// Mitsubishi GX Works2 project: 시퀀스 부분 반복 회로 예제   PLC: Q03UDV

PROGRAM MAIN
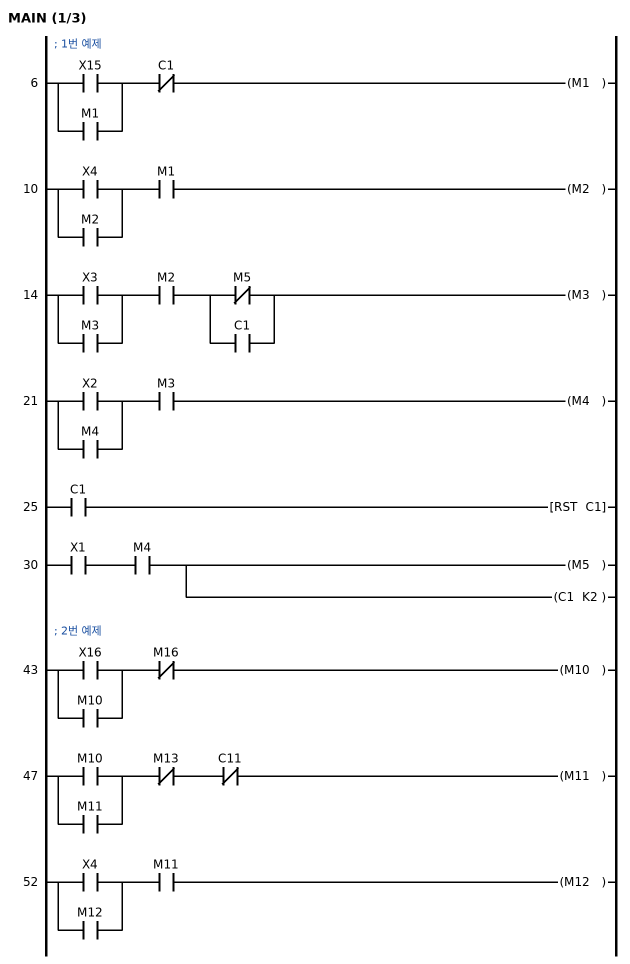
; 1번 예제
6     LD      X15
      OR      M1
      ANI     C1
      OUT     M1
10    LD      X4
      OR      M2
      AND     M1
      OUT     M2
14    LD      X3
      OR      M3
      AND     M2
      LDI     M5
      OR      C1
      ANB
      OUT     M3
21    LD      X2
      OR      M4
      AND     M3
      OUT     M4
25    LD      C1
      RST     C1
30    LD      X1
      AND     M4
      OUT     M5
      OUT     C1 K2
; 2번 예제
43    LD      X16
      OR      M10
      ANI     M16
      OUT     M10
47    LD      M10
      OR      M11
      ANI     M13
      ANI     C11
      OUT     M11
52    LD      X4
      OR      M12
      AND     M11
      OUT     M12
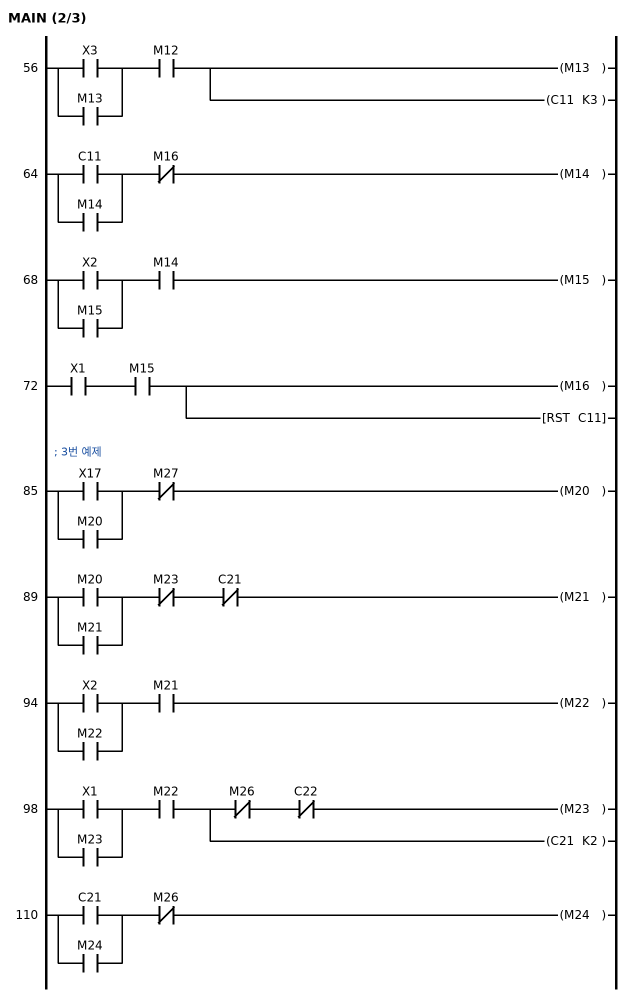
56    LD      X3
      OR      M13
      AND     M12
      OUT     M13
      OUT     C11 K3
64    LD      C11
      OR      M14
      ANI     M16
      OUT     M14
68    LD      X2
      OR      M15
      AND     M14
      OUT     M15
72    LD      X1
      AND     M15
      OUT     M16
      RST     C11
; 3번 예제
85    LD      X17
      OR      M20
      ANI     M27
      OUT     M20
89    LD      M20
      OR      M21
      ANI     M23
      ANI     C21
      OUT     M21
94    LD      X2
      OR      M22
      AND     M21
      OUT     M22
98    LD      X1
      OR      M23
      AND     M22
      MPS
      ANI     M26
      ANI     C22
      OUT     M23
      MPP
      OUT     C21 K2
110   LD      C21
      OR      M24
      ANI     M26
      OUT     M24
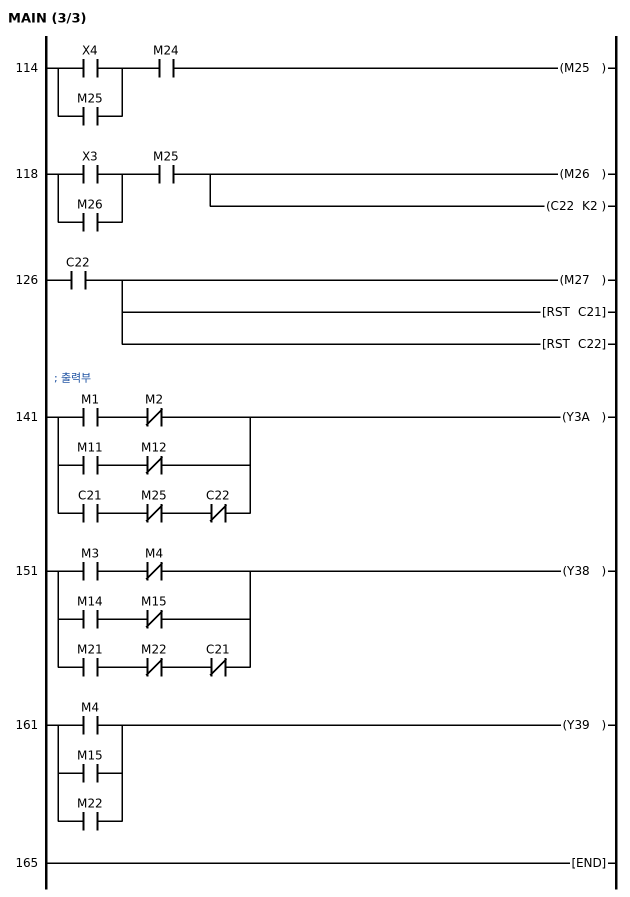
114   LD      X4
      OR      M25
      AND     M24
      OUT     M25
118   LD      X3
      OR      M26
      AND     M25
      OUT     M26
      OUT     C22 K2
126   LD      C22
      OUT     M27
      RST     C21
      RST     C22
; 출력부
141   LD      M1
      ANI     M2
      LD      M11
      ANI     M12
      ORB
      LD      C21
      ANI     M25
      ANI     C22
      ORB
      OUT     Y3A
151   LD      M3
      ANI     M4
      LD      M14
      ANI     M15
      ORB
      LD      M21
      ANI     M22
      ANI     C21
      ORB
      OUT     Y38
161   LD      M4
      OR      M15
      OR      M22
      OUT     Y39
165   END
END_PROGRAM
